TYPE MNG_POSE6 :(* position and orientation as an euler based pose *)
STRUCT
	x, y, z, a, b, c : REAL;
END_STRUCT
END_TYPE

(* stored: Version 1.1.0.1, ProductVersion 3.1.0.25
   DUT MNG_POSE6: Id {c443f680-1f9c-412c-a457-7cd5c7c4faf0} *)
